// TIA Portal V20 export
FUNCTION_BLOCK "FB_Recive_Water_Fountain_From_Rework"   // FB5, LAD
{ S7_Optimized_Access := 'TRUE' }
// stored: MemoryReserve 100, SetENOAutomatically false
   VAR_INPUT
      Emergency_Stop_Release : Bool;
      Start : Bool;
      Sensor_Water_Fountain_Before_Entrace_Functional_Test_Spinner_Conveyor_Belt : Bool;
      Sensor_Water_Fountain_Entrace_Functional_Test_Spinner_Conveyor_Belt : Bool;
      Sensor_Spinner_Entrace_Functional_Test_Position_Withdrawn : Bool;
      Sensor_Spinner_Entrace_Functional_Test_Position_Advanced : Bool;
      Sensor_Water_Fountain_Entrace_Functional_Test_After_Spinner_Conveyor_Belt : Bool;
      Sensor_Water_Fountain_Geting_Exit_Rework_Conveyor_Belt : Bool;
      Button_Water_Fountain_Get_Exit_Rework_Conveyor_Belt : Bool;
      Trigger_Read_Serial_Number_Entrace_Functional_Test : Bool;
   END_VAR
   VAR_OUTPUT
      Turn_On_Conveyor_Belt_Motor_Spinner_Get_Entrace_Function_Test : Bool;
      Valve_Advance_Spinner_Entrace_Functional_Test : Bool;
      Signal_Pre_Functional_Test_Production_Line : Bool;
   END_VAR
   VAR
      Aux_Trig_0 : Bool;
      Aux_Trig_1 : Bool;
      Aux_Trig_2 : Bool;
      Aux_Trig_3 : Bool;
      Aux_Trig_4 : Bool;
      Aux_Trig_5 : Bool;
      Aux_Trig_6 : Bool;
      Aux_Trig_7 : Bool;
      Aux_Trig_8 : Bool;
      Aux_Trig_9 : Bool;
      Button_Rework_Pressed : Bool;
      "Counter" : USInt;
      Timer_Delay_Turn_On_Motor_Spinner_Conveyor_Belt : TON_TIME;
      Counter_Water_Fountain_Entrace_Functional_Test { S7_SetPoint := 'True'} : CTUD_USINT;
   END_VAR
   VAR RETAIN
      Timer_Delay_Spin_Advanced { S7_SetPoint := 'True'} : TON_TIME;
   END_VAR
   VAR
      Timer_Delay_Spin_Withdrawn { S7_SetPoint := 'True'} : TON_TIME;
   END_VAR
   VAR_TEMP   // added for the SCL form of the ladder/FBD networks
      _w1 : Bool;
      _w2 : Bool;
   END_VAR
BEGIN

REGION Network 1
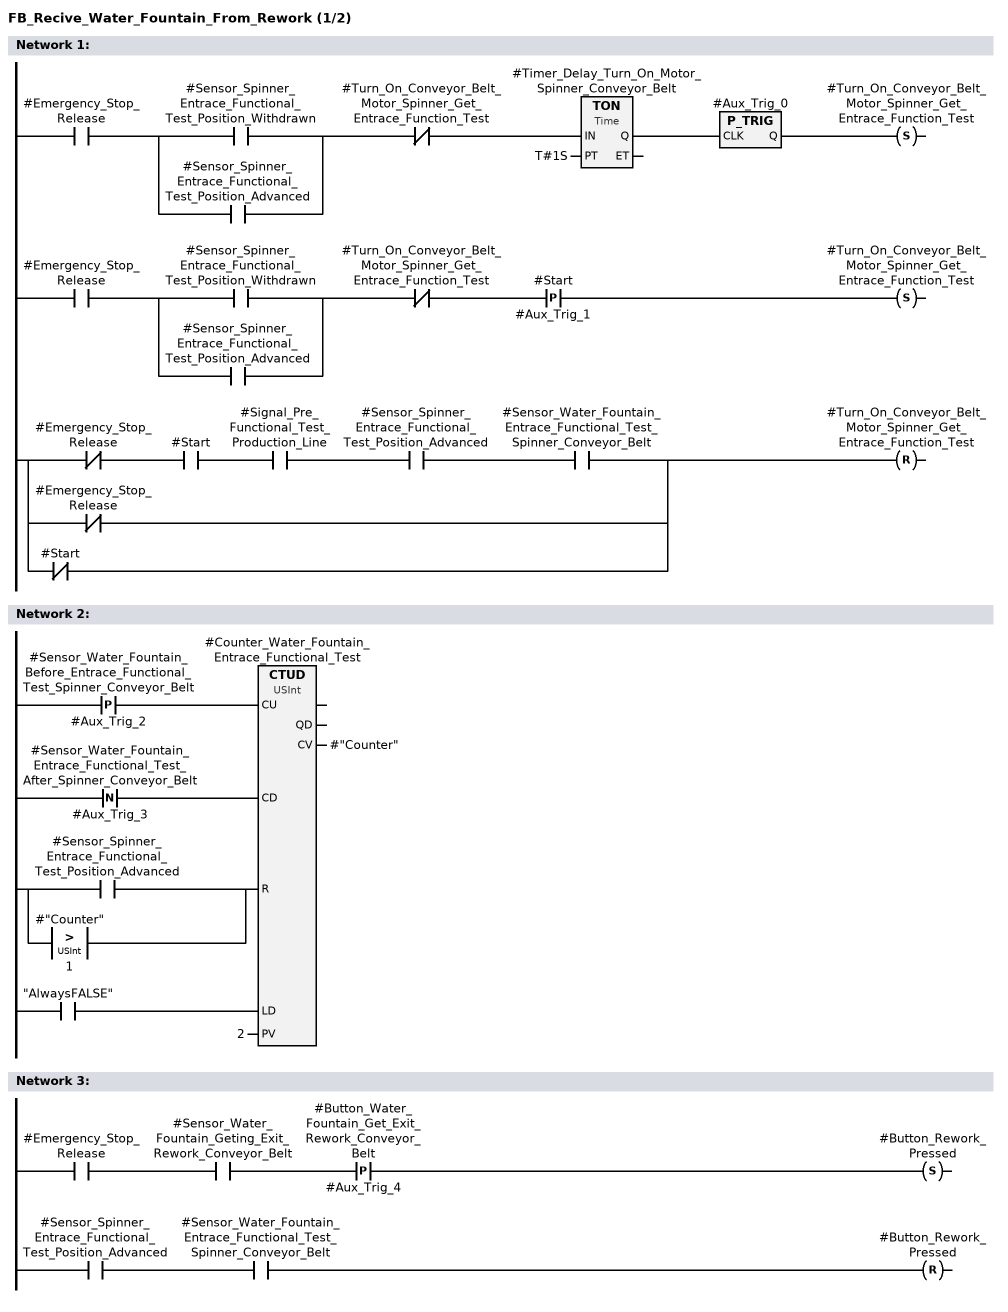
   RUNG wire#powerrail
      Contact( #Emergency_Stop_Release )
      wire#w1
      Contact( #Sensor_Spinner_Entrace_Functional_Test_Position_Withdrawn )
      wire#w2
      I_Contact( #Turn_On_Conveyor_Belt_Motor_Spinner_Get_Entrace_Function_Test )
      { S7_Templates := "time_type := Time" } #Timer_Delay_Turn_On_Motor_Spinner_Conveyor_Belt.TON(pt := T#1S, et =>)
      P_Trig( #Aux_Trig_0 )
      S_Coil( #Turn_On_Conveyor_Belt_Motor_Spinner_Get_Entrace_Function_Test )
   END_RUNG
   RUNG wire#w1
      Contact( #Sensor_Spinner_Entrace_Functional_Test_Position_Advanced )
   END_RUNG wire#w2
   RUNG wire#powerrail
      Contact( #Emergency_Stop_Release )
      wire#w3
      Contact( #Sensor_Spinner_Entrace_Functional_Test_Position_Withdrawn )
      wire#w4
      I_Contact( #Turn_On_Conveyor_Belt_Motor_Spinner_Get_Entrace_Function_Test )
      P_Contact(operand := #Start, bit := #Aux_Trig_1)
      S_Coil( #Turn_On_Conveyor_Belt_Motor_Spinner_Get_Entrace_Function_Test )
   END_RUNG
   RUNG wire#w3
      Contact( #Sensor_Spinner_Entrace_Functional_Test_Position_Advanced )
   END_RUNG wire#w4
   RUNG wire#powerrail
      I_Contact( #Emergency_Stop_Release )
      Contact( #Start )
      Contact( #Signal_Pre_Functional_Test_Production_Line )
      Contact( #Sensor_Spinner_Entrace_Functional_Test_Position_Advanced )
      Contact( #Sensor_Water_Fountain_Entrace_Functional_Test_Spinner_Conveyor_Belt )
      wire#w5
      R_Coil( #Turn_On_Conveyor_Belt_Motor_Spinner_Get_Entrace_Function_Test )
   END_RUNG
   RUNG wire#powerrail
      I_Contact( #Emergency_Stop_Release )
   END_RUNG wire#w5
   RUNG wire#powerrail
      I_Contact( #Start )
   END_RUNG wire#w5
   // the same network as SCL:
   #Timer_Delay_Turn_On_Motor_Spinner_Conveyor_Belt(IN := #Emergency_Stop_Release AND (#Sensor_Spinner_Entrace_Functional_Test_Position_Withdrawn OR #Sensor_Spinner_Entrace_Functional_Test_Position_Advanced) AND NOT #Turn_On_Conveyor_Belt_Motor_Spinner_Get_Entrace_Function_Test,   // TON
                           PT := T#1S);
   #_w1 := #Timer_Delay_Turn_On_Motor_Spinner_Conveyor_Belt.Q AND NOT #Aux_Trig_0;   // rising edge
   #Aux_Trig_0 := #Timer_Delay_Turn_On_Motor_Spinner_Conveyor_Belt.Q;
   IF #_w1 THEN #Turn_On_Conveyor_Belt_Motor_Spinner_Get_Entrace_Function_Test := TRUE; END_IF;
   #_w2 := #Emergency_Stop_Release AND (#Sensor_Spinner_Entrace_Functional_Test_Position_Withdrawn OR #Sensor_Spinner_Entrace_Functional_Test_Position_Advanced) AND NOT #Turn_On_Conveyor_Belt_Motor_Spinner_Get_Entrace_Function_Test AND #Start AND NOT #Aux_Trig_1;   // rising edge of #Start
   #Aux_Trig_1 := #Start;
   IF #_w2 THEN #Turn_On_Conveyor_Belt_Motor_Spinner_Get_Entrace_Function_Test := TRUE; END_IF;
   IF (NOT #Emergency_Stop_Release AND #Start AND #Signal_Pre_Functional_Test_Production_Line AND #Sensor_Spinner_Entrace_Functional_Test_Position_Advanced AND #Sensor_Water_Fountain_Entrace_Functional_Test_Spinner_Conveyor_Belt) OR NOT #Emergency_Stop_Release OR NOT #Start THEN
       #Turn_On_Conveyor_Belt_Motor_Spinner_Get_Entrace_Function_Test := FALSE;
   END_IF;
END_REGION

REGION Network 2
   RUNG wire#powerrail
      P_Contact(operand := #Sensor_Water_Fountain_Before_Entrace_Functional_Test_Spinner_Conveyor_Belt, bit := #Aux_Trig_2)
      { S7_Templates := "value_type := USInt" } #Counter_Water_Fountain_Entrace_Functional_Test.CTUD(cd := wire#w1, r := wire#w2, ld := wire#w3, pv := 2, qd =>, cv => #"Counter")
   END_RUNG
   RUNG wire#powerrail
      N_Contact(operand := #Sensor_Water_Fountain_Entrace_Functional_Test_After_Spinner_Conveyor_Belt, bit := #Aux_Trig_3)
   END_RUNG wire#w1
   RUNG wire#powerrail
      Contact( #Sensor_Spinner_Entrace_Functional_Test_Position_Advanced )
   END_RUNG wire#w2
   RUNG wire#powerrail
      { S7_Templates := "SrcType := USInt" } GT_Contact(in1 := #"Counter", in2 := 1)
   END_RUNG wire#w2
   RUNG wire#powerrail
      Contact( "AlwaysFALSE" )
   END_RUNG wire#w3
   // the same network as SCL:
   #_w1 := #Sensor_Water_Fountain_Before_Entrace_Functional_Test_Spinner_Conveyor_Belt AND NOT #Aux_Trig_2;   // rising edge of #Sensor_Water_Fountain_Before_Entrace_Functional_Test_Spinner_Conveyor_Belt
   #Aux_Trig_2 := #Sensor_Water_Fountain_Before_Entrace_Functional_Test_Spinner_Conveyor_Belt;
   #_w2 := NOT #Sensor_Water_Fountain_Entrace_Functional_Test_After_Spinner_Conveyor_Belt AND #Aux_Trig_3;   // falling edge of #Sensor_Water_Fountain_Entrace_Functional_Test_After_Spinner_Conveyor_Belt
   #Aux_Trig_3 := #Sensor_Water_Fountain_Entrace_Functional_Test_After_Spinner_Conveyor_Belt;
   #Counter_Water_Fountain_Entrace_Functional_Test(CU := #_w1,   // CTUD
                           CD := #_w2,
                           R := #Sensor_Spinner_Entrace_Functional_Test_Position_Advanced OR (#"Counter" > 1),
                           LD := "AlwaysFALSE",
                           PV := 2,
                           CV => #"Counter");
END_REGION

REGION Network 3
   RUNG wire#powerrail
      Contact( #Emergency_Stop_Release )
      Contact( #Sensor_Water_Fountain_Geting_Exit_Rework_Conveyor_Belt )
      P_Contact(operand := #Button_Water_Fountain_Get_Exit_Rework_Conveyor_Belt, bit := #Aux_Trig_4)
      S_Coil( #Button_Rework_Pressed )
   END_RUNG
   RUNG wire#powerrail
      Contact( #Sensor_Spinner_Entrace_Functional_Test_Position_Advanced )
      Contact( #Sensor_Water_Fountain_Entrace_Functional_Test_Spinner_Conveyor_Belt )
      R_Coil( #Button_Rework_Pressed )
   END_RUNG
   // the same network as SCL:
   #_w1 := #Emergency_Stop_Release AND #Sensor_Water_Fountain_Geting_Exit_Rework_Conveyor_Belt AND #Button_Water_Fountain_Get_Exit_Rework_Conveyor_Belt AND NOT #Aux_Trig_4;   // rising edge of #Button_Water_Fountain_Get_Exit_Rework_Conveyor_Belt
   #Aux_Trig_4 := #Button_Water_Fountain_Get_Exit_Rework_Conveyor_Belt;
   IF #_w1 THEN #Button_Rework_Pressed := TRUE; END_IF;
   IF #Sensor_Spinner_Entrace_Functional_Test_Position_Advanced AND #Sensor_Water_Fountain_Entrace_Functional_Test_Spinner_Conveyor_Belt THEN
       #Button_Rework_Pressed := FALSE;
   END_IF;
END_REGION

REGION Network 4
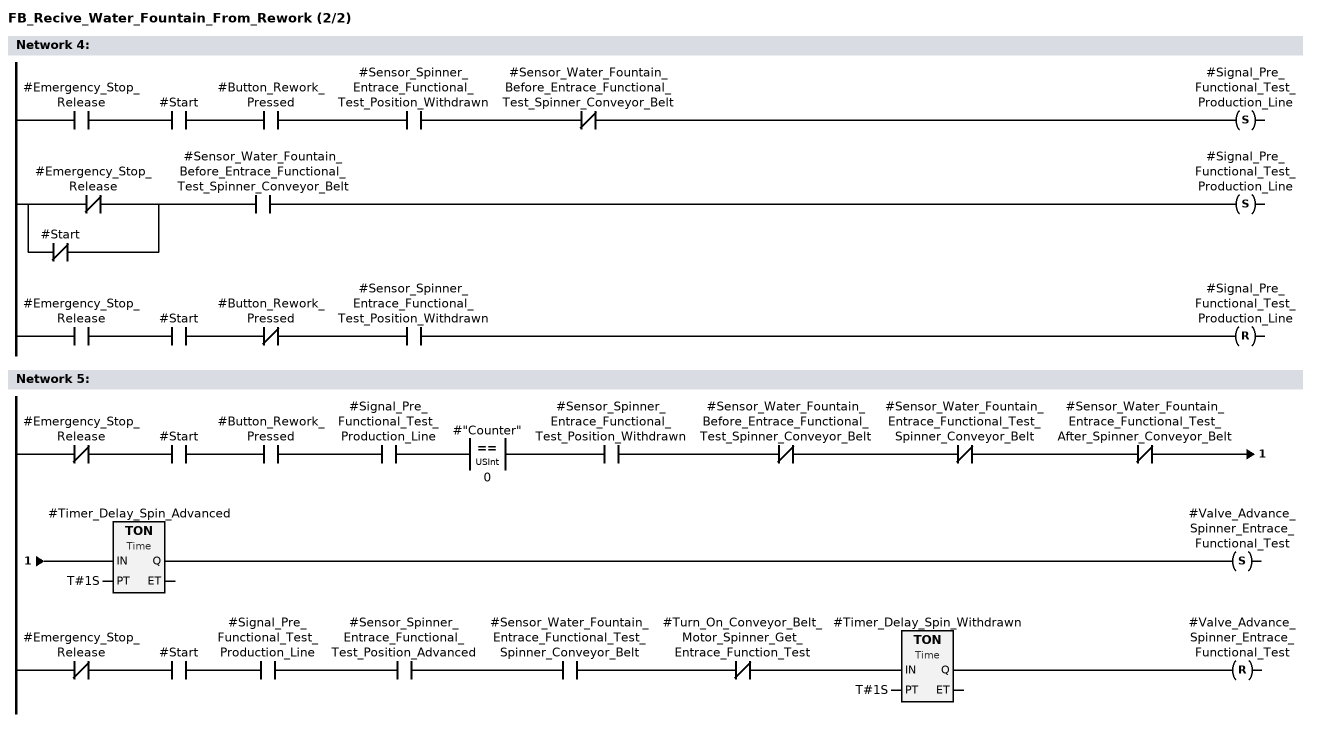
   RUNG wire#powerrail
      Contact( #Emergency_Stop_Release )
      Contact( #Start )
      Contact( #Button_Rework_Pressed )
      Contact( #Sensor_Spinner_Entrace_Functional_Test_Position_Withdrawn )
      I_Contact( #Sensor_Water_Fountain_Before_Entrace_Functional_Test_Spinner_Conveyor_Belt )
      S_Coil( #Signal_Pre_Functional_Test_Production_Line )
   END_RUNG
   RUNG wire#powerrail
      I_Contact( #Emergency_Stop_Release )
      wire#w1
      Contact( #Sensor_Water_Fountain_Before_Entrace_Functional_Test_Spinner_Conveyor_Belt )
      S_Coil( #Signal_Pre_Functional_Test_Production_Line )
   END_RUNG
   RUNG wire#powerrail
      I_Contact( #Start )
   END_RUNG wire#w1
   RUNG wire#powerrail
      Contact( #Emergency_Stop_Release )
      Contact( #Start )
      I_Contact( #Button_Rework_Pressed )
      Contact( #Sensor_Spinner_Entrace_Functional_Test_Position_Withdrawn )
      R_Coil( #Signal_Pre_Functional_Test_Production_Line )
   END_RUNG
   // the same network as SCL:
   IF #Emergency_Stop_Release AND #Start AND #Button_Rework_Pressed AND #Sensor_Spinner_Entrace_Functional_Test_Position_Withdrawn AND NOT #Sensor_Water_Fountain_Before_Entrace_Functional_Test_Spinner_Conveyor_Belt THEN
       #Signal_Pre_Functional_Test_Production_Line := TRUE;
   END_IF;
   IF (NOT #Emergency_Stop_Release OR NOT #Start) AND #Sensor_Water_Fountain_Before_Entrace_Functional_Test_Spinner_Conveyor_Belt THEN
       #Signal_Pre_Functional_Test_Production_Line := TRUE;
   END_IF;
   IF #Emergency_Stop_Release AND #Start AND NOT #Button_Rework_Pressed AND #Sensor_Spinner_Entrace_Functional_Test_Position_Withdrawn THEN
       #Signal_Pre_Functional_Test_Production_Line := FALSE;
   END_IF;
END_REGION

REGION Network 5
   RUNG wire#powerrail
      I_Contact( #Emergency_Stop_Release )
      Contact( #Start )
      Contact( #Button_Rework_Pressed )
      Contact( #Signal_Pre_Functional_Test_Production_Line )
      { S7_Templates := "SrcType := USInt" } EQ_Contact(in1 := #"Counter", in2 := 0)
      Contact( #Sensor_Spinner_Entrace_Functional_Test_Position_Withdrawn )
      I_Contact( #Sensor_Water_Fountain_Before_Entrace_Functional_Test_Spinner_Conveyor_Belt )
      I_Contact( #Sensor_Water_Fountain_Entrace_Functional_Test_Spinner_Conveyor_Belt )
      I_Contact( #Sensor_Water_Fountain_Entrace_Functional_Test_After_Spinner_Conveyor_Belt )
      { S7_Templates := "time_type := Time" } #Timer_Delay_Spin_Advanced.TON(pt := T#1S, et =>)
      S_Coil( #Valve_Advance_Spinner_Entrace_Functional_Test )
   END_RUNG
   RUNG wire#powerrail
      I_Contact( #Emergency_Stop_Release )
      Contact( #Start )
      Contact( #Signal_Pre_Functional_Test_Production_Line )
      Contact( #Sensor_Spinner_Entrace_Functional_Test_Position_Advanced )
      Contact( #Sensor_Water_Fountain_Entrace_Functional_Test_Spinner_Conveyor_Belt )
      I_Contact( #Turn_On_Conveyor_Belt_Motor_Spinner_Get_Entrace_Function_Test )
      { S7_Templates := "time_type := Time" } #Timer_Delay_Spin_Withdrawn.TON(pt := T#1S, et =>)
      R_Coil( #Valve_Advance_Spinner_Entrace_Functional_Test )
   END_RUNG
   // the same network as SCL:
   #Timer_Delay_Spin_Advanced(IN := NOT #Emergency_Stop_Release AND #Start AND #Button_Rework_Pressed AND #Signal_Pre_Functional_Test_Production_Line AND (#"Counter" = 0) AND #Sensor_Spinner_Entrace_Functional_Test_Position_Withdrawn AND NOT #Sensor_Water_Fountain_Before_Entrace_Functional_Test_Spinner_Conveyor_Belt AND NOT #Sensor_Water_Fountain_Entrace_Functional_Test_Spinner_Conveyor_Belt AND NOT #Sensor_Water_Fountain_Entrace_Functional_Test_After_Spinner_Conveyor_Belt,   // TON
                           PT := T#1S);
   IF #Timer_Delay_Spin_Advanced.Q THEN #Valve_Advance_Spinner_Entrace_Functional_Test := TRUE; END_IF;
   #Timer_Delay_Spin_Withdrawn(IN := NOT #Emergency_Stop_Release AND #Start AND #Signal_Pre_Functional_Test_Production_Line AND #Sensor_Spinner_Entrace_Functional_Test_Position_Advanced AND #Sensor_Water_Fountain_Entrace_Functional_Test_Spinner_Conveyor_Belt AND NOT #Turn_On_Conveyor_Belt_Motor_Spinner_Get_Entrace_Function_Test,   // TON
                           PT := T#1S);
   IF #Timer_Delay_Spin_Withdrawn.Q THEN #Valve_Advance_Spinner_Entrace_Functional_Test := FALSE; END_IF;
END_REGION
END_FUNCTION_BLOCK
